FUNCTION_BLOCK LOG_X (* Composite FB wrapping other FBs *)
  (* Standard: 61499-2 *)
  (* Version 1.0, 2021-08-05, dorofeev *)
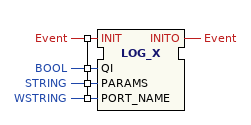
  EVENT_INPUT
    INIT WITH PORT_NAME, PARAMS, QI; (* Initialization Request *)
  END_EVENT
  EVENT_OUTPUT
    INITO;
  END_EVENT
  VAR_INPUT
    QI : BOOL; (* Input event qualifier *)
    PARAMS : STRING;
    PORT_NAME : WSTRING;
  END_VAR
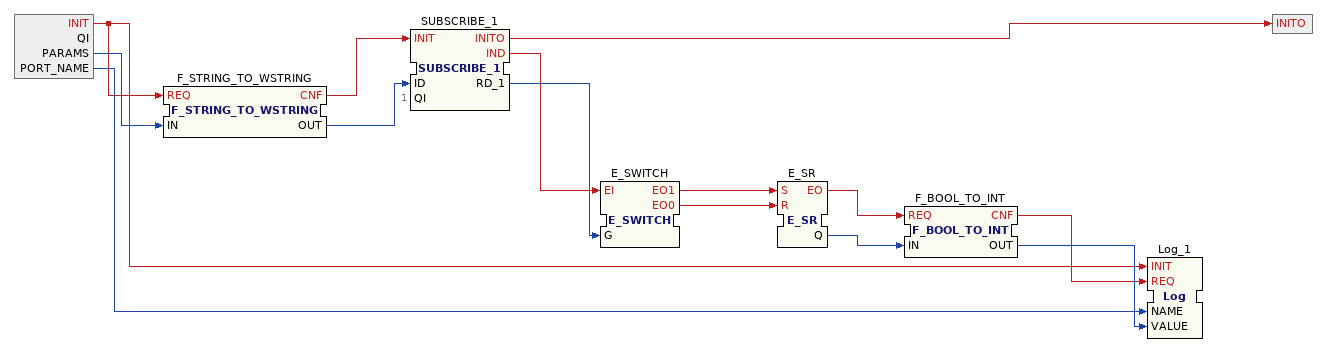
  FBS
    F_STRING_TO_WSTRING : F_STRING_TO_WSTRING;
    SUBSCRIBE_1 : SUBSCRIBE_1(QI := 1);
    Log_1 : Log;
    E_SWITCH : E_SWITCH;
    E_SR : E_SR;
    F_BOOL_TO_INT : F_BOOL_TO_INT;
  END_FBS
  EVENT_CONNECTIONS
    INIT TO F_STRING_TO_WSTRING.REQ;
    F_STRING_TO_WSTRING.CNF TO SUBSCRIBE_1.INIT;
    SUBSCRIBE_1.INITO TO INITO;
    INIT TO Log_1.INIT;
    E_SWITCH.EO1 TO E_SR.S;
    E_SWITCH.EO0 TO E_SR.R;
    SUBSCRIBE_1.IND TO E_SWITCH.EI;
    E_SR.EO TO F_BOOL_TO_INT.REQ;
    F_BOOL_TO_INT.CNF TO Log_1.REQ;
  END_CONNECTIONS
  DATA_CONNECTIONS
    PARAMS TO F_STRING_TO_WSTRING.IN;
    F_STRING_TO_WSTRING.OUT TO SUBSCRIBE_1.ID;
    SUBSCRIBE_1.RD_1 TO E_SWITCH.G;
    E_SR.Q TO F_BOOL_TO_INT.IN;
    F_BOOL_TO_INT.OUT TO Log_1.VALUE;
    PORT_NAME TO Log_1.NAME;
  END_CONNECTIONS
END_FUNCTION_BLOCK
